(* Logix 5000 project; controller WINDPLC vendor 1 type 14 code 106 rev 28.12; software revision 28.03 *)

TASK MainTask (continuous, watchdog 500 ms) : MainProgram
TASK PID (periodic, rate 10 ms, priority 1, watchdog 500 ms) : VFDWindSpeed

MODULES
   Local : vendor 1 type 14 code 106 (Compact 0, rev 28.12)
      WINDTUNNEL : 1734-AENTR (Ethernet 192.168.1.12, rev 6.11, Output RPI 20 ms)   // Wind Tunnel Project
         DRIFTANDLIFT : 1734-IE2V (PointIO 2, rev 3.5, Input RPI 80 ms)   // Dirft and lift sensors
         PRESSUREANDDIAL : 1734-IE2V (PointIO 1, rev 3.4, Input RPI 80 ms)   // Pressure sensor and dial
         BUTTONINPUT : 1734-IB8 (PointIO 4, rev 3.30)   // Buttons
         VFDOUTPUT : 1734-OE2V (PointIO 3, rev 3.9, Output RPI 80 ms)   // VFD Output Module
         BUTTONOUTPUT : 1734-OB8 (PointIO 5, rev 3.22)   // Button Outputs
END_MODULES

VAR_GLOBAL   (* controller tags *)
   AIRDENSITY : REAL := 1.293; {constant}   // Air density
   CurrentState : DINT;   // Current State
   DataViewScreenButton : ALIAS FOR WINDTUNNEL:4:I.2;   // Dataview Button Screen
   DRAGCAPACITY : REAL := 227.0; {constant}   // Drag Capacity
   DRAGSENSITIVITY : REAL := 10.0; {constant}   // Drag Sensitivity
   GRAMFORCETONEWTONS : REAL := 0.00980665; {constant}   // Gram Force To Newtons
   HMI_ACKNOWLEDGE_BTN : BOOL;   // Emergency button acknowledgement
   HMI_Actual_WindSpeed : REAL;   // The actual windspeed inside the windtunnel
   HMI_DATAVIEWER : BOOL := 1;   // HMI Data Viewer Screen
   HMI_Desired_WindSpeed : REAL := 9.0;   // The users desired windspeed
   HMI_Drag : REAL;   // Drag force output in Newtons
   HMI_EMERGENCY_ESTOP : ALIAS FOR WINDTUNNEL:4:I.6;   // Emergency Stop
   HMI_EXTRACTUSB : BOOL := 1;   // HMI Extraction USB
   HMI_Forces_Graph_Max_Range : DINT;   // adjusts the max range of the forces graph
   HMI_Forces_Graph_TimeSpan : DINT;   // adjusts the timespan of the forces graph
   HMI_KDERIVATIVE : DINT;   // Derivative Constant for PID
   HMI_KINTEGRAL : DINT;   // Intregal Constant for PID
   HMI_KPOSITION : DINT;   // Proportional Constant for PID
   HMI_Lift : REAL;   // Lift Output in Newtons
   HMI_MANUAL_TOGGLE : BOOL;   // Manual Override
   HMI_Pressure : REAL;   // Pressure output in Pascals
   HMI_START : BOOL;   // Digital Start Button
   HMI_STOP : BOOL;   // Digital Stop Button
   HMI_WindSpeed_Graph_Max_Range : DINT;   // adjusts the max range for wind-speed graph
   HMI_WindSpeed_Graph_TimeSpan : DINT;   // adjusts the timespand of the wind-speed graph
   HMI_WINDSPEED_SLIDER : INT;   // SLIDER
   HMI_WindSpeedToggle : BOOL;   // HMI_WindSpeedToggle
   HMI_WindVelocity : REAL;   // Wind Velocity
   HMIVFDInput : ALIAS FOR WINDTUNNEL:3:O.Ch0Data;   // Input voltage to the VFD
   InputDragSensor : ALIAS FOR WINDTUNNEL:1:I.Ch1Data;   // Input Drag Sensor
   InputLiftSensor : ALIAS FOR WINDTUNNEL:2:I.Ch0Data;   // Input Lift Sensor
   InputPressureSensor : ALIAS FOR WINDTUNNEL:1:I.Ch0Data;   // Input Pressure Sensor
   LIFTCAPACITY : REAL := 454.0; {constant}   // Lift Capacity
   LIFTSENSITIVITY : REAL := 10.0; {constant}   // Lift Sensitivity
   MILLIVOLTSTOVOLTS : REAL := 1000.0; {constant}   // Millivolts to Volts
   MULTIPLYBY2 : REAL := 2.0; {constant}   // Multiply by 2
   NextState : DINT;   // Next State
   PanelButtonStart : ALIAS FOR WINDTUNNEL:4:I.0;   // Start Button
   PanelButtonStop : ALIAS FOR WINDTUNNEL:4:I.1;   // Pannel Stop Button
   PRESSUREGAIN : REAL := 125.0; {constant}   // Pressure Gain
   ToggleLight : ALIAS FOR WINDTUNNEL:5:O.0;   // Toggle Light
   USBExtractionButton : ALIAS FOR WINDTUNNEL:4:I.3;   // USB Extraction Button
   WindSpeedDial : ALIAS FOR WINDTUNNEL:2:I.Ch1Data;   // Wind Speed Dial
END_VAR

PROGRAM MainProgram   (* main routine MainRoutine, fault routine FaultDetection *)

ROUTINE DragSensor   (* structured text *)
// Drag Sensor Calculation
   /******************************************************************************
    * Name: DragSensor
    * Description: Drag Sensor Calculation
    *
    * Arguments: none
    * Return: None
    *
    * Author: Leland Dean, Carolyn Richards, Noah Gastelum
    * Date: Feb 21, 2025
    * Modified Data: N/A
    *****************************************************************************/
   HMI_Drag [:=] ((InputDragSensor / MILLIVOLTSTOVOLTS) / DRAGSENSITIVITY) * DRAGCAPACITY * GRAMFORCETONEWTONS;
END_ROUTINE

ROUTINE FaultDetection   (* structured text *)
// Fault recovery
   //HMI_ACKNOWLEDGE
END_ROUTINE

ROUTINE LiftSensor   (* structured text *)
// Lift Sensor Calculation
   /******************************************************************************
    * Name: LiftSensor
    * Description: Lift Sensor Calculation
    *
    * Arguments: none
    * Return: None
    *
    * Author: Leland Dean, Carolyn Richards, Noah Gastelum
    * Date: Feb 21, 2025
    * Modified Data: N/A
    *****************************************************************************/
   HMI_Lift [:=] ((InputLiftSensor/ MILLIVOLTSTOVOLTS) / LIFTSENSITIVITY) * LIFTCAPACITY * GRAMFORCETONEWTONS;
END_ROUTINE

ROUTINE MainRoutine   (* structured text *)
   /******************************************************************************
    * Name: MainRoutine
    * Description: Main routine to call other routines
    *
    * Arguments: none
    * Return: None
    *
    * Author: Leland Dean, Carolyn Richards, Noah Gastelum
    * Date: Feb 21, 2025
    * Modified Data: N/A
    *****************************************************************************/
   JSR(WindTunnelMainLogic);
   
END_ROUTINE

ROUTINE PressureSensor   (* structured text *)
// Pressure Sensor Calculation
   /******************************************************************************
    * Name: PressureSensor
    * Description: Pressure Sensor Calculation
    *
    * Arguments: none
    * Return: None
    *
    * Author: Leland Dean, Carolyn Richards, Noah Gastelum
    * Date: Feb 21, 2025
    * Modified Data: N/A
    *****************************************************************************/
   HMI_Pressure [:=] InputPressureSensor / MILLIVOLTSTOVOLTS * PRESSUREGAIN;
END_ROUTINE

ROUTINE WindTunnelMainLogic   (* structured text *)
   /******************************************************************************
    * Name: WindTunnelMainLogic
    * Description: Wind Tunnel State Machine
    *
    * Arguments: none
    * Return: None
    *
    * Author: Leland Dean, Carolyn Richards, Noah Gastelum
    * Date: Feb 21, 2025
    * Modified Data: N/A
    *****************************************************************************/
   IF S:FS THEN
   	CurrentState := 0;
   	NextState := 0;
   	HMI_Desired_WindSpeed := 9.00;
   	HMI_Forces_Graph_Max_Range := 5;
   	HMI_WindSpeed_Graph_Max_Range := 650;
   	HMI_KPOSITION := 600.0;
   	HMI_KINTEGRAL := 1.0;
   	HMI_KDERIVATIVE := 0.0;
   END_IF;
   
   IF DataViewScreenButton AND NOT HMI_EMERGENCY_ESTOP AND NOT HMI_ACKNOWLEDGE_BTN THEN
   	HMI_DATAVIEWER := 1;
   ELSE
   	HMI_DATAVIEWER := 0;
   END_IF;
   
   IF USBExtractionButton AND NOT HMI_EMERGENCY_ESTOP AND NOT HMI_ACKNOWLEDGE_BTN THEN
   	HMI_EXTRACTUSB := 1;
   
   ELSE
   	HMI_EXTRACTUSB := 0;
   END_IF;
   
   IF HMI_EMERGENCY_ESTOP THEN
   	HMIVFDInput := 0;
   	ToggleLight := 1;
   	NextState := 100;
   ELSE
   	ToggleLight := 0;
   END_IF;
   
   
   IF CurrentState <> NextState THEN
   	CurrentState := NextState;
   END_IF;
   
   CASE CurrentState OF
   
   	0: /* INIT State */
   		IF HMI_START OR PanelButtonStart THEN
   			NextState := 1;
   			HMIVFDInput := 0;
   		END_IF;
   
   	1: /* ON State */
   		jsr(PressureSensor);
   		jsr(LiftSensor);
   		jsr(DragSensor);
   
   
   	  	IF HMI_STOP OR PanelButtonStop THEN
   			HMIVFDInput := 0;
   	  		NextState := 0;
   	  	END_IF;
   
   		IF HMI_MANUAL_TOGGLE THEN
   			HMIVFDInput := HMI_WINDSPEED_SLIDER;
   		ELSE
   			IF HMI_WindSpeedToggle THEN
   				IF HMI_Desired_WindSpeed < 9.00 THEN
   					HMI_Desired_WindSpeed := 9.00;
   				ELSIF HMI_Desired_WindSpeed > 30.00 THEN
   					HMI_Desired_WindSpeed := 30.00;
   				END_IF;
   			ELSE
   				HMI_Desired_WindSpeed := (30.00 - 9.00) / (10561 - 4) *  WindSpeedDial + 9.0;
   			END_IF;
   		END_IF;
   
   	100:
   		IF NOT HMI_EMERGENCY_ESTOP AND HMI_ACKNOWLEDGE_BTN THEN
   			NextState := 0;
   			ToggleLight := 0;
   		END_IF;
   
   END_CASE;
   
   
   
   
   
   
END_ROUTINE
END_PROGRAM

PROGRAM VFDWindSpeed   (* main routine WindSpeedTask *)
VAR
   derivativeError : REAL;   // Calculated derivative error
   integralError : REAL;   // Calculated integral error
   posError : REAL;   // Calculated Proportional error
   preError : REAL;   // Previous Proportional Error
END_VAR

ROUTINE WindSpeed   (* structured text *)
// WindSpeed Calculation
   /******************************************************************************
    * Name: WindSpeed
    * Description: Wind Speed Calculation
    *
    * Arguments: none
    * Return: None
    *
    * Author: Leland Dean, Carolyn Richards, Noah Gastelum
    * Date: Feb 21, 2025
    * Modified Data: N/A
    *****************************************************************************/
   HMI_Actual_WindSpeed [:=] sqrt((MULTIPLYBY2*(InputPressureSensor / MILLIVOLTSTOVOLTS * PRESSUREGAIN))/AIRDENSITY);
END_ROUTINE

ROUTINE WindSpeedMainLogic   (* structured text *)
   /******************************************************************************
    * Name: WindSpeedMainLogic
    * Description: Wind Speed Logic for different task states.
    *
    * Arguments: none
    * Return: None
    *
    * Author: Leland Dean, Carolyn Richards, Noah Gastelum
    * Date: Feb 21, 2025
    * Modified Data: N/A
    *****************************************************************************/
   IF HMI_EMERGENCY_ESTOP OR HMI_ACKNOWLEDGE_BTN OR HMI_STOP OR PanelButtonStop THEN
   	HMIVFDInput := 0;
   	posError := 0;
   	preError := 0;
   	integralError := 0;
   	derivativeError := 0;
   	HMI_MANUAL_TOGGLE := 0;
   	HMI_WINDSPEED_SLIDER := 0;
   
   
   ELSIF HMI_MANUAL_TOGGLE THEN
   	posError := 0;
   	preError := 0;
   	integralError := 0;
   	derivativeError := 0;
   
   ELSIF CurrentState = 1 THEN
   	JSR(WindSpeed);
   
   	posError := HMI_Desired_WindSpeed - HMI_Actual_WindSpeed;
   	integralError := integralError + posError;
   	derivativeError := posError - preError;
   	preError := posError;
   	HMIVFDInput := HMI_KPOSITION * posError + HMI_KINTEGRAL * integralError + HMI_KDERIVATIVE * derivativeError;
   
   ELSE
   	HMIVFDInput := 0;
   	posError := 0;
   	integralError := 0;
   	derivativeError := 0;
   	preError := 0;
   END_IF;
   
   
END_ROUTINE

ROUTINE WindSpeedTask   (* structured text *)
   /******************************************************************************
    * Name: WindSpeedTask
    * Description: Wind Speed Task call routine to call other routines
    *
    * Arguments: none
    * Return: None
    *
    * Author: Leland Dean, Carolyn Richards, Noah Gastelum
    * Date: Feb 21, 2025
    * Modified Data: N/A
    *****************************************************************************/
   JSR(WindSpeedMainLogic);
   
END_ROUTINE
END_PROGRAM
